{attribute 'linkalways'} 
{attribute 'no_explicit_call' := 'This FB is a CLASS and must be accessed using methods or properties'}
{attribute 'enable_dynamic_creation'}
FUNCTION_BLOCK NodeFactory IMPLEMENTS I_NodeFactory
VAR
	prototypeHost : NodePrototypeHost;
END_VAR

METHOD PUBLIC Accept
VAR_INPUT
	Visitor : I_NodeFactoryVisitor;
END_VAR
Visitor.VisitNodeFactory(this^);
END_METHOD

METHOD AddNodeAsPrototype : I_NodePrototype
VAR_INPUT
	Path : T_MAXSTRING;
	Node : I_Node;
END_VAR
AddNodeAsPrototype := prototypeHost.AddNodeAsPrototype(Path, Node);
END_METHOD

METHOD PUBLIC AddNodePrototype
VAR_INPUT
	NodePrototype : I_NodePrototype;
END_VAR
prototypeHost.AddNodePrototype(NodePrototype);
END_METHOD

METHOD PUBLIC InstallNodePack
VAR_INPUT
	NodePack : I_NodePack;
END_VAR
NodePack.RegisterWithNodeFactory(This^);
END_METHOD

PROPERTY PUBLIC NodePrototypes : I_NodePrototypes
GET
NodePrototypes := prototypeHost;
END_GET
END_PROPERTY

METHOD PUBLIC TryCreateNodeByType : BOOL
VAR_INPUT
	Path : T_MAXSTRING;
	Destination : REFERENCE TO I_Node;
END_VAR
VAR
	nodePrototype : I_NodePrototype;
END_VAR
IF NOT prototypeHost.TryGetNodePrototypeByPath(Path, nodePrototype) THEN
	RETURN;
END_IF

Destination := nodePrototype.Clone();
TryCreateNodeByType := TRUE;
END_METHOD

END_FUNCTION_BLOCK

(* stored: Version 1.1.0.1, ProductVersion 3.1.4024.12
   POU NodeFactory: Id {3a71411c-013f-04b4-2fdb-abd75ba10395}, SpecialFunc None
   Method Accept: Id {513e8062-8019-4c39-a286-8ae6858476b0}
   Method AddNodeAsPrototype: Id {6b2e8ed8-096f-49b5-9cbd-63b800d603fb}
   Method AddNodePrototype: Id {8bdcf9b9-8b58-40a1-ac90-376fd07e397c}
   Method InstallNodePack: Id {0ec00c43-b35f-0669-2893-bc57927b1baa}
   Property NodePrototypes: Id {6e589d04-a62a-451e-86c4-f664af7187bb}
   Get Get: Id {461b6771-5200-47c5-b4a0-772c4681a403}
   Method TryCreateNodeByType: Id {ceb4bb2e-8751-4cf7-92a9-b7b5faf2cfa2} *)
